FUNCTION_BLOCK FEED_AJUST (* Sets feed in m/s and can multiply it to a fraction of the original value *)
  (* Standard: 61499-2 *)
  (* Version 1.0, 09-01-12, Guilherme Jarentchuk, Universidade do Estado de Santa Catarina *)
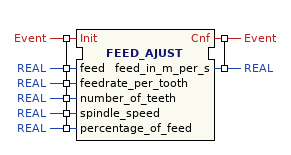
  EVENT_INPUT
    Init WITH feed, feedrate_per_tooth, number_of_teeth, spindle_speed, percentage_of_feed; (* Initialization event *)
  END_EVENT
  EVENT_OUTPUT
    Cnf WITH feed_in_m_per_s; (* Execution complete *)
  END_EVENT
  VAR_INPUT
    feed : REAL := 0; (* Axes resultant speed in m/s *)
    feedrate_per_tooth : REAL := 0; (* In mm *)
    number_of_teeth : REAL := 0;
    spindle_speed : REAL := 0; (* In rotations/s *)
    percentage_of_feed : REAL := 100;
  END_VAR
  VAR_OUTPUT
    feed_in_m_per_s : REAL; (* Resultant axes linear speed in m/s *)
  END_VAR
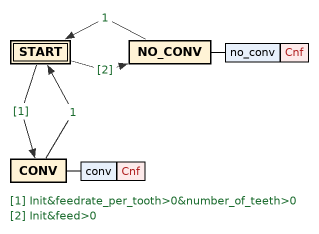
  EC_STATES
    START; (* Initial state *)
    NO_CONV : no_conv -> Cnf; (* Without unit convertion *)
    CONV : conv -> Cnf; (* With unit convertion *)
  END_STATES
  EC_TRANSITIONS
    START TO NO_CONV := Init&feed>0;
    NO_CONV TO START := 1;
    START TO CONV := Init&feedrate_per_tooth>0&number_of_teeth>0;
    CONV TO START := 1;
  END_TRANSITIONS
  ALGORITHM conv IN Lua: (* Convert feed unit and apply percentage *)
feed_in_m_per_s = feedrate_per_tooth*number_of_teeth*spindle_speed
feed_in_m_per_s = (percentage_of_feed/100)*feed_in_m_per_s
  END_ALGORITHM
  ALGORITHM no_conv IN Lua: (* Just apply percentage *)
feed_in_m_per_s = (percentage_of_feed/100)*feed
  END_ALGORITHM
END_FUNCTION_BLOCK
